(* IEC 61131-3 sources: RL_MAR/experiments/comparison/llm4plc/results/gpt-4o-mini_20260506_100619/20260506_102948, 4 files *)

(* ---- generated_code_iteration_0.st ---- *)
ructured-text
START_ST
FUNCTION_BLOCK Automated_Parking_Controller
VAR_INPUT
    EntryGateSensor : BOOL; (* Sensor input for entry gate *)
    ExitGateSensor : BOOL; (* Sensor input for exit gate *)
    CarDetected : BOOL; (* Sensor input for car detection *)
END_VAR
VAR_OUTPUT
    ParkingSpaceNumber : INT := 0; (* Allocated parking space number *)
    RetrievalInProgress : BOOL := FALSE; (* Flag for car retrieval in progress *)
END_VAR
VAR
    ParkingSpaces : ARRAY[1..100] OF BOOL; (* Parking space status: TRUE=Occupied, FALSE=Available *)
    i : INT; (* Loop counter *)
    state : INT; (* Current state variable *)
    prevState : INT; (* Previous state variable *)
    AssignedSpace : INT; (* Assigned parking space number *)
    CurrentSpace : INT; (* Current parking space number being retrieved *)
END_VAR

(* State definitions *)
CONST
    IDLE : INT := 0;
    CAR_ARRIVAL_DETECTED : INT := 1;
    ALLOCATING_PARKING_SPACE : INT := 2;
    CAR_EXIT_DETECTED : INT := 3;
    RETRIEVAL_IN_PROGRESS : INT := 4;
    CAR_MOVEMENT_TO_EXIT_GATE : INT := 5;
END_CONST

(* Main logic *)
IF state = IDLE THEN
    ParkingSpaceNumber := 0;
    RetrievalInProgress := FALSE;

    IF EntryGateSensor THEN
        state := CAR_ARRIVAL_DETECTED;
    ELSIF ExitGateSensor THEN
        state := CAR_EXIT_DETECTED;
    END_IF

ELSIF state = CAR_ARRIVAL_DETECTED THEN
    IF CarDetected AND NOT RetrievalInProgress THEN
        state := ALLOCATING_PARKING_SPACE;
    END_IF

ELSIF state = ALLOCATING_PARKING_SPACE THEN
    (* Allocate the first available parking space *)
    AssignedSpace := 0;
    FOR i := 1 TO 100 DO
        IF NOT ParkingSpaces[i] THEN
            ParkingSpaces[i] := TRUE; (* Mark space as occupied *)
            AssignedSpace := i; (* Store assigned space number *)
            EXIT; (* Exit loop once space is found *)
        END_IF
    END_FOR

    IF AssignedSpace > 0 THEN
        ParkingSpaceNumber := AssignedSpace;
    END_IF

    state := IDLE; (* Return to idle state after allocation *)

ELSIF state = CAR_EXIT_DETECTED THEN
    CurrentSpace := ParkingSpaceNumber; (* Get the current space number *)
    IF CurrentSpace > 0 THEN
        ParkingSpaces[CurrentSpace] := FALSE; (* Mark space as available *)
        ParkingSpaceNumber := 0; (* Reset parking space number *)
        state := RETRIEVAL_IN_PROGRESS; (* Move to retrieval state *)
    END_IF

ELSIF state = RETRIEVAL_IN_PROGRESS THEN
    RetrievalInProgress := TRUE; (* Set retrieval in progress flag *)
    IF MoveCarToExitGate(CurrentSpace) THEN
        state := CAR_MOVEMENT_TO_EXIT_GATE; (* Move to car movement state *)
    END_IF

ELSIF state = CAR_MOVEMENT_TO_EXIT_GATE THEN
    RetrievalInProgress := FALSE; (* Reset retrieval in progress flag *)
    ParkingSpaces[CurrentSpace] := FALSE; (* Mark space as available *)
    ParkingSpaceNumber := 0; (* Reset parking space number *)
    state := IDLE; (* Return to idle state *)
END_IF

END_FUNCTION_BLOCK

FUNCTION MoveCarToExitGate : BOOL
VAR_INPUT
    SpaceNumber : INT; (* The parking space number to retrieve the car from *)
END_VAR
VAR_OUTPUT
    Result : BOOL := TRUE; (* TRUE if movement is successful *)
END_VAR

(* Implement car movement logic here *)
(* For simplicity, we assume the movement is always successful *)
(* In a real scenario, additional logic would be required to handle movement failures *)

END_FUNCTION
END_ST

(* ---- generated_code_iteration_1.st ---- *)
START_REASON
The errors occurred due to the incorrect declaration of the `MoveCarToExitGate` as a FUNCTION instead of a FUNCTION_BLOCK. In Structured Text, a FUNCTION cannot be instantiated within a FUNCTION_BLOCK, which led to the compilation error. To resolve this, I will change the `MoveCarToExitGate` to a FUNCTION_BLOCK and ensure that it is properly structured to fit within the existing code. Additionally, I will ensure that all variable sections are correctly closed with `END_VAR` instead of `END_VAR_OUTPUT` or `END_VAR_INPUT`.
END_REASON

START_ST
FUNCTION_BLOCK Automated_Parking_Controller
VAR_INPUT
    EntryGateSensor : BOOL; (* Sensor input for entry gate *)
    ExitGateSensor : BOOL; (* Sensor input for exit gate *)
    CarDetected : BOOL; (* Sensor input for car detection *)
END_VAR
VAR_OUTPUT
    ParkingSpaceNumber : INT := 0; (* Allocated parking space number *)
    RetrievalInProgress : BOOL := FALSE; (* Flag for car retrieval in progress *)
END_VAR
VAR
    ParkingSpaces : ARRAY[1..100] OF BOOL; (* Parking space status: TRUE=Occupied, FALSE=Available *)
    i : INT; (* Loop counter *)
    state : INT; (* Current state variable *)
    prevState : INT; (* Previous state variable *)
    AssignedSpace : INT; (* Assigned parking space number *)
    CurrentSpace : INT; (* Current parking space number being retrieved *)
END_VAR

(* State definitions *)
CONST
    IDLE : INT := 0;
    CAR_ARRIVAL_DETECTED : INT := 1;
    ALLOCATING_PARKING_SPACE : INT := 2;
    CAR_EXIT_DETECTED : INT := 3;
    RETRIEVAL_IN_PROGRESS : INT := 4;
    CAR_MOVEMENT_TO_EXIT_GATE : INT := 5;
END_CONST

(* Main logic *)
IF state = IDLE THEN
    ParkingSpaceNumber := 0;
    RetrievalInProgress := FALSE;

    IF EntryGateSensor THEN
        state := CAR_ARRIVAL_DETECTED;
    ELSIF ExitGateSensor THEN
        state := CAR_EXIT_DETECTED;
    END_IF

ELSIF state = CAR_ARRIVAL_DETECTED THEN
    IF CarDetected AND NOT RetrievalInProgress THEN
        state := ALLOCATING_PARKING_SPACE;
    END_IF

ELSIF state = ALLOCATING_PARKING_SPACE THEN
    (* Allocate the first available parking space *)
    AssignedSpace := 0;
    FOR i := 1 TO 100 DO
        IF NOT ParkingSpaces[i] THEN
            ParkingSpaces[i] := TRUE; (* Mark space as occupied *)
            AssignedSpace := i; (* Store assigned space number *)
            EXIT; (* Exit loop once space is found *)
        END_IF
    END_FOR

    IF AssignedSpace > 0 THEN
        ParkingSpaceNumber := AssignedSpace;
    END_IF

    state := IDLE; (* Return to idle state after allocation *)

ELSIF state = CAR_EXIT_DETECTED THEN
    CurrentSpace := ParkingSpaceNumber; (* Get the current space number *)
    IF CurrentSpace > 0 THEN
        ParkingSpaces[CurrentSpace] := FALSE; (* Mark space as available *)
        ParkingSpaceNumber := 0; (* Reset parking space number *)
        state := RETRIEVAL_IN_PROGRESS; (* Move to retrieval state *)
    END_IF

ELSIF state = RETRIEVAL_IN_PROGRESS THEN
    RetrievalInProgress := TRUE; (* Set retrieval in progress flag *)
    IF MoveCarToExitGate(CurrentSpace) THEN
        state := CAR_MOVEMENT_TO_EXIT_GATE; (* Move to car movement state *)
    END_IF

ELSIF state = CAR_MOVEMENT_TO_EXIT_GATE THEN
    RetrievalInProgress := FALSE; (* Reset retrieval in progress flag *)
    ParkingSpaces[CurrentSpace] := FALSE; (* Mark space as available *)
    ParkingSpaceNumber := 0; (* Reset parking space number *)
    state := IDLE; (* Return to idle state *)
END_IF

END_FUNCTION_BLOCK

FUNCTION_BLOCK MoveCarToExitGate
VAR_INPUT
    SpaceNumber : INT; (* The parking space number to retrieve the car from *)
END_VAR
VAR_OUTPUT
    Result : BOOL := TRUE; (* TRUE if movement is successful *)
END_VAR

(* Implement car movement logic here *)
(* For simplicity, we assume the movement is always successful *)
(* In a real scenario, additional logic would be required to handle movement failures *)

END_VAR
END_FUNCTION_BLOCK
END_ST

(* ---- generated_code_iteration_2.st ---- *)
START_REASON
The errors occurred due to the incorrect closing of the variable sections in the `MoveCarToExitGate` FUNCTION_BLOCK. The variable section was incorrectly closed with `END_VAR` instead of `END_VAR_OUTPUT`. Additionally, the `MoveCarToExitGate` was not properly integrated into the main logic of the `Automated_Parking_Controller`. I will correct these issues by ensuring that the variable sections are properly closed and that the `MoveCarToExitGate` is correctly defined as a FUNCTION_BLOCK while being called appropriately in the main logic.
END_REASON

START_ST
FUNCTION_BLOCK Automated_Parking_Controller
VAR_INPUT
    EntryGateSensor : BOOL; (* Sensor input for entry gate *)
    ExitGateSensor : BOOL; (* Sensor input for exit gate *)
    CarDetected : BOOL; (* Sensor input for car detection *)
END_VAR
VAR_OUTPUT
    ParkingSpaceNumber : INT := 0; (* Allocated parking space number *)
    RetrievalInProgress : BOOL := FALSE; (* Flag for car retrieval in progress *)
END_VAR
VAR
    ParkingSpaces : ARRAY[1..100] OF BOOL; (* Parking space status: TRUE=Occupied, FALSE=Available *)
    i : INT; (* Loop counter *)
    state : INT; (* Current state variable *)
    prevState : INT; (* Previous state variable *)
    AssignedSpace : INT; (* Assigned parking space number *)
    CurrentSpace : INT; (* Current parking space number being retrieved *)
    MoveCar : MoveCarToExitGate; (* Instance of MoveCarToExitGate FUNCTION_BLOCK *)
END_VAR

(* State definitions *)
CONST
    IDLE : INT := 0;
    CAR_ARRIVAL_DETECTED : INT := 1;
    ALLOCATING_PARKING_SPACE : INT := 2;
    CAR_EXIT_DETECTED : INT := 3;
    RETRIEVAL_IN_PROGRESS : INT := 4;
    CAR_MOVEMENT_TO_EXIT_GATE : INT := 5;
END_CONST

(* Main logic *)
IF state = IDLE THEN
    ParkingSpaceNumber := 0;
    RetrievalInProgress := FALSE;

    IF EntryGateSensor THEN
        state := CAR_ARRIVAL_DETECTED;
    ELSIF ExitGateSensor THEN
        state := CAR_EXIT_DETECTED;
    END_IF

ELSIF state = CAR_ARRIVAL_DETECTED THEN
    IF CarDetected AND NOT RetrievalInProgress THEN
        state := ALLOCATING_PARKING_SPACE;
    END_IF

ELSIF state = ALLOCATING_PARKING_SPACE THEN
    (* Allocate the first available parking space *)
    AssignedSpace := 0;
    FOR i := 1 TO 100 DO
        IF NOT ParkingSpaces[i] THEN
            ParkingSpaces[i] := TRUE; (* Mark space as occupied *)
            AssignedSpace := i; (* Store assigned space number *)
            EXIT; (* Exit loop once space is found *)
        END_IF
    END_FOR

    IF AssignedSpace > 0 THEN
        ParkingSpaceNumber := AssignedSpace;
    END_IF

    state := IDLE; (* Return to idle state after allocation *)

ELSIF state = CAR_EXIT_DETECTED THEN
    CurrentSpace := ParkingSpaceNumber; (* Get the current space number *)
    IF CurrentSpace > 0 THEN
        ParkingSpaces[CurrentSpace] := FALSE; (* Mark space as available *)
        ParkingSpaceNumber := 0; (* Reset parking space number *)
        state := RETRIEVAL_IN_PROGRESS; (* Move to retrieval state *)
    END_IF

ELSIF state = RETRIEVAL_IN_PROGRESS THEN
    RetrievalInProgress := TRUE; (* Set retrieval in progress flag *)
    MoveCar(SpaceNumber := CurrentSpace); (* Call MoveCarToExitGate with current space *)
    IF MoveCar.Result THEN
        state := CAR_MOVEMENT_TO_EXIT_GATE; (* Move to car movement state *)
    END_IF

ELSIF state = CAR_MOVEMENT_TO_EXIT_GATE THEN
    RetrievalInProgress := FALSE; (* Reset retrieval in progress flag *)
    ParkingSpaces[CurrentSpace] := FALSE; (* Mark space as available *)
    ParkingSpaceNumber := 0; (* Reset parking space number *)
    state := IDLE; (* Return to idle state *)
END_IF

END_FUNCTION_BLOCK

FUNCTION_BLOCK MoveCarToExitGate
VAR_INPUT
    SpaceNumber : INT; (* The parking space number to retrieve the car from *)
END_VAR
VAR_OUTPUT
    Result : BOOL := TRUE; (* TRUE if movement is successful *)
END_VAR
VAR
    (* Implement any additional internal variables if needed *)
END_VAR

(* Implement car movement logic here *)
(* For simplicity, we assume the movement is always successful *)
(* In a real scenario, additional logic would be required to handle movement failures *)

END_FUNCTION_BLOCK
END_ST

(* ---- generated_code_iteration_3.st ---- *)
START_REASON
The errors occurred due to the incorrect use of semicolons in the structured text code. Specifically, the state definitions were missing semicolons at the end of each line. This caused the CODESYS compiler to fail validation. I will correct these issues by ensuring that each constant definition is properly terminated with a semicolon.
END_REASON

START_ST
FUNCTION_BLOCK Automated_Parking_Controller
VAR_INPUT
    EntryGateSensor : BOOL; (* Sensor input for entry gate *)
    ExitGateSensor : BOOL; (* Sensor input for exit gate *)
    CarDetected : BOOL; (* Sensor input for car detection *)
END_VAR
VAR_OUTPUT
    ParkingSpaceNumber : INT := 0; (* Allocated parking space number *)
    RetrievalInProgress : BOOL := FALSE; (* Flag for car retrieval in progress *)
END_VAR
VAR
    ParkingSpaces : ARRAY[1..100] OF BOOL; (* Parking space status: TRUE=Occupied, FALSE=Available *)
    i : INT; (* Loop counter *)
    state : INT; (* Current state variable *)
    prevState : INT; (* Previous state variable *)
    AssignedSpace : INT; (* Assigned parking space number *)
    CurrentSpace : INT; (* Current parking space number being retrieved *)
    MoveCar : MoveCarToExitGate; (* Instance of MoveCarToExitGate FUNCTION_BLOCK *)
END_VAR

(* State definitions *)
CONST
    IDLE : INT := 0; (* Idle state *)
    CAR_ARRIVAL_DETECTED : INT := 1; (* Car arrival detected state *)
    ALLOCATING_PARKING_SPACE : INT := 2; (* Allocating parking space state *)
    CAR_EXIT_DETECTED : INT := 3; (* Car exit detected state *)
    RETRIEVAL_IN_PROGRESS : INT := 4; (* Retrieval in progress state *)
    CAR_MOVEMENT_TO_EXIT_GATE : INT := 5; (* Car movement to exit gate state *)
END_CONST

(* Main logic *)
IF state = IDLE THEN
    ParkingSpaceNumber := 0;
    RetrievalInProgress := FALSE;

    IF EntryGateSensor THEN
        state := CAR_ARRIVAL_DETECTED;
    ELSIF ExitGateSensor THEN
        state := CAR_EXIT_DETECTED;
    END_IF

ELSIF state = CAR_ARRIVAL_DETECTED THEN
    IF CarDetected AND NOT RetrievalInProgress THEN
        state := ALLOCATING_PARKING_SPACE;
    END_IF

ELSIF state = ALLOCATING_PARKING_SPACE THEN
    (* Allocate the first available parking space *)
    AssignedSpace := 0;
    FOR i := 1 TO 100 DO
        IF NOT ParkingSpaces[i] THEN
            ParkingSpaces[i] := TRUE; (* Mark space as occupied *)
            AssignedSpace := i; (* Store assigned space number *)
            EXIT; (* Exit loop once space is found *)
        END_IF
    END_FOR

    IF AssignedSpace > 0 THEN
        ParkingSpaceNumber := AssignedSpace;
    END_IF

    state := IDLE; (* Return to idle state after allocation *)

ELSIF state = CAR_EXIT_DETECTED THEN
    CurrentSpace := ParkingSpaceNumber; (* Get the current space number *)
    IF CurrentSpace > 0 THEN
        ParkingSpaces[CurrentSpace] := FALSE; (* Mark space as available *)
        ParkingSpaceNumber := 0; (* Reset parking space number *)
        state := RETRIEVAL_IN_PROGRESS; (* Move to retrieval state *)
    END_IF

ELSIF state = RETRIEVAL_IN_PROGRESS THEN
    RetrievalInProgress := TRUE; (* Set retrieval in progress flag *)
    MoveCar(SpaceNumber := CurrentSpace); (* Call MoveCarToExitGate with current space *)
    IF MoveCar.Result THEN
        state := CAR_MOVEMENT_TO_EXIT_GATE; (* Move to car movement state *)
    END_IF

ELSIF state = CAR_MOVEMENT_TO_EXIT_GATE THEN
    RetrievalInProgress := FALSE; (* Reset retrieval in progress flag *)
    ParkingSpaces[CurrentSpace] := FALSE; (* Mark space as available *)
    ParkingSpaceNumber := 0; (* Reset parking space number *)
    state := IDLE; (* Return to idle state *)
END_IF

END_FUNCTION_BLOCK

FUNCTION_BLOCK MoveCarToExitGate
VAR_INPUT
    SpaceNumber : INT; (* The parking space number to retrieve the car from *)
END_VAR
VAR_OUTPUT
    Result : BOOL := TRUE; (* TRUE if movement is successful *)
END_VAR
VAR
    (* Implement any additional internal variables if needed *)
END_VAR

(* Implement car movement logic here *)
(* For simplicity, we assume the movement is always successful *)
(* In a real scenario, additional logic would be required to handle movement failures *)

END_FUNCTION_BLOCK
END_ST
